// TIA Portal V18 export
TYPE "WriteProcessData"
// stored: IsFailsafeCompliant false
   STRUCT
      AssemblyResult1 : Byte;
      AssemblyResult2 : Byte;
      StartForce1 : Real;
      StartLVDT1 : Real;
      ProcessForce1 : Real;
      ProcessLVDT1 : Real;
      EndForce1 : Real;
      EndLVDT1 : Real;
      StartForce2 : Real;
      StartLVDT2 : Real;
      ProcessForce2 : Real;
      ProcessLVDT2 : Real;
      EndForce2 : Real;
      EndLVDT2 : Real;
   END_STRUCT;
END_TYPE
